// TIA Portal V17 export
// export: Created 2024-08-07T21:44:12.5687433Z, ExportSetting WithDefaults, DisplayName Totally Integrated Automation Portal, DisplayVersion V17 Update 7, DisplayName TIA Portal Openness, DisplayVersion V17 Update 7, DisplayName TIA Portal Version Control Interface, DisplayVersion V17, DisplayName SINAMICS Startdrive Advanced, DisplayVersion V17 SP2, DisplayName SINAMICS Startdrive G110M, G120, G120C, G120D, G120P, G115D, DisplayVersion V17 SP2, DisplayName SINAMICS Startdrive G130, G150, S120, S150, SINAMICS MV, S210, DisplayVersion V17 SP2, DisplayName STEP 7 Professional, DisplayVersion V17 Update 7, DisplayName STEP 7 Safety, DisplayVersion V17 Update 6, DisplayName WinCC Advanced / Unified PC, DisplayVersion V17 Update 7
VAR_GLOBAL   // PLC tag table "system"
   Clock_Byte AT %MB0 : Byte;
   Clock_10Hz AT %M0.0 : Bool;
   Clock_5Hz AT %M0.1 : Bool;
   "Clock_2.5Hz" AT %M0.2 : Bool;
   Clock_2Hz AT %M0.3 : Bool;
   "Clock_1.25Hz" AT %M0.4 : Bool;
   Clock_1Hz AT %M0.5 : Bool;
   "Clock_0.625Hz" AT %M0.6 : Bool;
   "Clock_0.5Hz" AT %M0.7 : Bool;
   System_Byte AT %MB1 : Byte;
   FirstScan AT %M1.0 : Bool;
   DiagStatusUpdate AT %M1.1 : Bool;
   AlwaysTRUE AT %M1.2 : Bool;
   AlwaysFALSE AT %M1.3 : Bool;
END_VAR
